{attribute 'qualified_only'}
VAR_GLOBAL CONSTANT
	/// Fifo overhead needed to manage the string buffer
	FifoOverhead : UDINT := 10;

	/// Buffer size of temporary buffer used to persist all log messages in one cycle. 
	BufferSize : UDINT := (100 * (Tc2_System.MAX_STRING_LENGTH + FifoOverhead));
END_VAR

(* stored: Version 1.1.0.1
   GVL Constants: Id {6adae184-6d3f-480d-9baa-dc87732a07ab}, ParameterList True *)
